Staubli VAL3: sendRosMsg.pgx

public program sendRosMsg(sio& x_sTcpSocket (dimensions=1), Prefix& x_pPrefix (dimensions=1), Header& x_hHeader (dimensions=1), Body& x_bBody (dimensions=1), num& x_nConnFlag (dimensions=1))
begin
  // Copyright (c) 2016, Ocado Technology - Robotics Research Team
  //
  // Licensed under the Apache License, Version 2.0 (the "License");
  // you may not use this file except in compliance with the License.
  // You may obtain a copy of the License at
  //
  //     http://www.apache.org/licenses/LICENSE-2.0
  //
  // Unless required by applicable law or agreed to in writing, software
  // distributed under the License is distributed on an "AS IS" BASIS,
  // WITHOUT WARRANTIES OR CONDITIONS OF ANY KIND, either express or implied.
  // See the License for the specific language governing permissions and
  // limitations under the License.



  call sendData(x_sTcpSocket,x_pPrefix.nData,x_nConnFlag)
  call sendData(x_sTcpSocket,x_hHeader.nData,x_nConnFlag)
  call sendData(x_sTcpSocket,x_bBody.nData,x_nConnFlag)
end
